FUNCTION_BLOCK D_OUT (* Service Interface Function Block Type *)
  (* Standard: 61499-2 *)
  (* Version 1.0, 2023-12-12, filipe *)
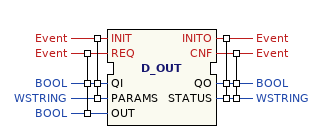
  EVENT_INPUT
    INIT WITH QI, PARAMS; (* Service Initialization *)
    REQ WITH QI, OUT; (* Service Request *)
  END_EVENT
  EVENT_OUTPUT
    INITO WITH QO, STATUS; (* Initialization Confirm *)
    CNF WITH QO, STATUS; (* Confirmation of Requested Service *)
  END_EVENT
  VAR_INPUT
    QI : BOOL := TRUE; (* Event Input Qualifier *)
    PARAMS : WSTRING; (* Service Parameters *)
    OUT : BOOL;
  END_VAR
  VAR_OUTPUT
    QO : BOOL; (* Event Output Qualifier *)
    STATUS : WSTRING; (* Service Status *)
  END_VAR
  (* Service /: Service Interface Function Block Type *)
END_FUNCTION_BLOCK
